FUNCTION_BLOCK FB_ESSMonitoringMCU5001a EXTENDS FB_ESSMonitoringBase
VAR
    //Outputs
    {attribute 'TcLinkTo' := 'TIID^Device 2 (EtherCAT)^KF201 (EK1100)^KF208 (EL2014)^DIG Outputs^Channel 1^Output'}
    bStatusLED AT %Q*: BOOL;
    {attribute 'TcLinkTo' := 'TIID^Device 2 (EtherCAT)^KF201 (EK1100)^KF207 (EL2014)^DIG Outputs^Channel 4^Output'}
    bAcknowledgeLED AT %Q*: BOOL;
    {attribute 'TcLinkTo' := 'TIID^Device 2 (EtherCAT)^KF201 (EK1100)^KF208 (EL2014)^DIG Outputs^Channel 2^Output'}
    bEStopLED AT %Q*: BOOL;
    {attribute 'TcLinkTo' := 'TIID^Device 2 (EtherCAT)^KF201 (EK1100)^KF208 (EL2014)^DIG Outputs^Channel 4^Output'}
    bErrorLED AT %Q*: BOOL;

    //Inputs
    {attribute 'TcLinkTo' := 'TIID^Device 2 (EtherCAT)^KF201 (EK1100)^KF204 (EL1808)^Channel 1^Input'}
    b24VDC1_OK AT %I*: BOOL;
    {attribute 'TcLinkTo' := 'TIID^Device 2 (EtherCAT)^KF201 (EK1100)^KF204 (EL1808)^Channel 2^Input'}
    b24VDC2_OK AT %I*: BOOL;
    {attribute 'TcLinkTo' := 'TIID^Device 2 (EtherCAT)^KF201 (EK1100)^KF204 (EL1808)^Channel 3^Input'}
    b24VDC3_OK AT %I*: BOOL;
    {attribute 'TcLinkTo' := 'TIID^Device 2 (EtherCAT)^KF201 (EK1100)^KF204 (EL1808)^Channel 4^Input'}
    b48VDC1_OK AT %I*: BOOL;
    {attribute 'TcLinkTo' := 'TIID^Device 2 (EtherCAT)^KF201 (EK1100)^KF204 (EL1808)^Channel 5^Input'}
    b48VDC2_OK AT %I*: BOOL;
    {attribute 'TcLinkTo' := 'TIID^Device 2 (EtherCAT)^KF201 (EK1100)^KF204 (EL1808)^Channel 6^Input'}
    b48VDC3_OK AT %I*: BOOL;
    {attribute 'TcLinkTo' := 'TIID^Device 2 (EtherCAT)^KF201 (EK1100)^KF204 (EL1808)^Channel 7^Input'}
    b48VDC4_OK AT %I*: BOOL;
    {attribute 'TcLinkTo' := 'TIID^Device 2 (EtherCAT)^KF201 (EK1100)^KF203 (EL1808)^Channel 1^Input'}
    bFuse1_OK AT %I*: BOOL;
    {attribute 'TcLinkTo' := 'TIID^Device 2 (EtherCAT)^KF201 (EK1100)^KF203 (EL1808)^Channel 2^Input'}
    bFuse2_Error AT %I*: BOOL;
    {attribute 'TcLinkTo' := 'TIID^Device 2 (EtherCAT)^KF201 (EK1100)^KF203 (EL1808)^Channel 3^Input'}
    bFuse3_Error AT %I*: BOOL;
    {attribute 'TcLinkTo' := 'TIID^Device 2 (EtherCAT)^KF201 (EK1100)^KF203 (EL1808)^Channel 4^Input'}
    bFuse4_OK AT %I*: BOOL;
    {attribute 'TcLinkTo' := 'TIID^Device 2 (EtherCAT)^KF201 (EK1100)^KF203 (EL1808)^Channel 5^Input'}
    bFuse5_OK AT %I*: BOOL;
    {attribute 'TcLinkTo' := 'TIID^Device 2 (EtherCAT)^KF201 (EK1100)^KF203 (EL1808)^Channel 6^Input'}
    bFuse6_OK AT %I*: BOOL;
    {attribute 'TcLinkTo' := 'TIID^Device 2 (EtherCAT)^KF201 (EK1100)^KF203 (EL1808)^Channel 7^Input'}
    bFuse7_OK AT %I*: BOOL;
    {attribute 'TcLinkTo' := 'TIID^Device 2 (EtherCAT)^KF201 (EK1100)^KF203 (EL1808)^Channel 8^Input'}
    bFuse8_OK AT %I*: BOOL;
    {attribute 'TcLinkTo' := 'TIID^Device 2 (EtherCAT)^KF201 (EK1100)^KF205 (EL1808)^Channel 1^Input'}
    bEStopReleased AT %I*: BOOL;
    {attribute 'TcLinkTo' := 'TIID^Device 2 (EtherCAT)^KF201 (EK1100)^KF205 (EL1808)^Channel 2^Input'}
    bSTOReleased AT %I*: BOOL;
    {attribute 'TcLinkTo' := 'TIID^Device 2 (EtherCAT)^KF201 (EK1100)^KF206 (EL1808)^Channel 2^Input'}
    bMCBFan_OK AT %I*: BOOL;
    {attribute 'TcLinkTo' := 'TIID^Device 2 (EtherCAT)^KF201 (EK1100)^KF206 (EL1808)^Channel 3^Input'}
    bSPD_OK AT %I*: BOOL;
    {attribute 'TcLinkTo' := 'TIID^Device 2 (EtherCAT)^KF201 (EK1100)^KF206 (EL1808)^Channel 4^Input'}
    bDoorClosed AT %I*: BOOL;
    {attribute 'TcLinkTo' := 'TIID^Device 2 (EtherCAT)^KF201 (EK1100)^KF205 (EL1808)^Channel 8^Input'}
    bAcknowledgeButton AT %I*: BOOL;
    {attribute 'TcLinkTo' := 'TIID^Device 2 (EtherCAT)^KF201 (EK1100)^KF209 (EL3214)^RTD Inputs Channel 1^Value'}
    nTemp1 AT %I*: INT;
    {attribute 'TcLinkTo' := 'TIID^Device 2 (EtherCAT)^KF201 (EK1100)^KF209 (EL3214)^RTD Inputs Channel 2^Value'}
    nTemp2 AT %I*: INT;
    {attribute 'TcLinkTo' := 'TIID^Device 2 (EtherCAT)^KF201 (EK1100)^KF209 (EL3214)^RTD Inputs Channel 3^Value'}
    nTemp3 AT %I*: INT;
    {attribute 'TcLinkTo' := 'TIID^Device 2 (EtherCAT)^KF201 (EK1100)^KF209 (EL3214)^RTD Inputs Channel 4^Value'}
    nTemp4 AT %I*: INT;
    {attribute 'TcLinkTo' := 'TIID^Device 2 (EtherCAT)^Inputs^DevState'}
    nEcMasterDevState AT %I*: UINT;
END_VAR

SUPER^();

METHOD mLink
// Input variables
AcknowledgeButton := bAcknowledgeButton;
EcMasterDevState := nEcMasterDevState;

// Output variables
bAcknowledgeLED := AcknowledgeLED;
bStatusLED := StatusLED;
bEStopLED := EStopLED;
bErrorLED := ErrorLED;

IF iSafetyProvider <> 0 AND_THEN iSafetyProvider.P_ReadFromSafetyController THEN
    _EStopReleased := iSafetyProvider.P_EStopOK;
    _STOReleased := iSafetyProvider.P_STO_OK;
ELSE
    _EStopReleased := bEStopReleased;
    _STOReleased := bSTOReleased;
END_IF;

EStopReleased := _EStopReleased;
END_METHOD

METHOD mSetResetAlarmsLeds
VAR_INST
    index: UINT;
    aDeadBandActive: ARRAY [1..4] OF BOOL;
    nDeadBandTemperature: INT := 3;
    aTemperatureAlarm: ARRAY [1..4] OF BOOL;
END_VAR
mSetReset(stAlarmList := aAlarmList[1], bOk := b24VDC1_OK);
mSetReset(stAlarmList := aAlarmList[2], bOk := b24VDC2_OK);
mSetReset(stAlarmList := aAlarmList[3], bOk := b24VDC3_OK);

mSetReset(stAlarmList := aAlarmList[4], bOk := b48VDC1_OK);
mSetReset(stAlarmList := aAlarmList[5], bOk := b48VDC2_OK);
mSetReset(stAlarmList := aAlarmList[6], bOk := b48VDC3_OK);
mSetReset(stAlarmList := aAlarmList[7], bOk := b48VDC4_OK);

mSetReset(stAlarmList := aAlarmList[8], bOk := bMCBFan_OK);
mSetReset(stAlarmList := aAlarmList[9], bOk := bSPD_OK);
mSetReset(stAlarmList := aAlarmList[10], bOk := bDoorClosed);

mSetReset(stAlarmList := aAlarmList[11], bOk := bFuse1_OK);
mSetReset(stAlarmList := aAlarmList[12], bOk := NOT bFuse2_Error);
mSetReset(stAlarmList := aAlarmList[13], bOk := NOT bFuse3_Error);
mSetReset(stAlarmList := aAlarmList[14], bOk := bFuse4_OK);
mSetReset(stAlarmList := aAlarmList[15], bOk := bFuse5_OK);
mSetReset(stAlarmList := aAlarmList[16], bOk := bFuse6_OK);
mSetReset(stAlarmList := aAlarmList[17], bOk := bFuse7_OK);
mSetReset(stAlarmList := aAlarmList[18], bOk := bFuse8_OK);

mSetReset(stAlarmList := aAlarmList[19], bOk := EStopReleased);

mSetReset(stAlarmList := aAlarmList[24], bOk := NOT bEcMasterError);
mSetReset(stAlarmList := aAlarmList[25], bOk := NOT bSlaveStateNotOP);
mSetReset(stAlarmList := aAlarmList[26], bOk := NOT bSlaveLinkError);
mSetReset(stAlarmList := aAlarmList[27], bOk := NOT bCycleTimeExceeded);
mSetReset(stAlarmList := aAlarmList[28], bOk := NOT bCPUOverloaded);


aTemperatureAlarm[1] :=
    nTemp1 > nMAX_TEMP
    OR (aDeadBandActive[1] AND nTemp1 > (nMAX_TEMP - nDeadBandTemperature));
aDeadBandActive[1] := aTemperatureAlarm[1];
mSetReset(stAlarmList := aAlarmList[20], bOk := NOT aTemperatureAlarm[1]);

aTemperatureAlarm[2] :=
    nTemp2 > nMAX_TEMP
    OR (aDeadBandActive[2] AND nTemp2 > (nMAX_TEMP - nDeadBandTemperature));
aDeadBandActive[2] := aTemperatureAlarm[2];
mSetReset(stAlarmList := aAlarmList[21], bOk := NOT aTemperatureAlarm[2]);

aTemperatureAlarm[3] :=
    nTemp3 > nMAX_TEMP
    OR (aDeadBandActive[3] AND nTemp3 > (nMAX_TEMP - nDeadBandTemperature));
aDeadBandActive[3] := aTemperatureAlarm[3];
mSetReset(stAlarmList := aAlarmList[22], bOk := NOT aTemperatureAlarm[3]);

aTemperatureAlarm[4] :=
    nTemp4 > nMAX_TEMP
    OR (aDeadBandActive[4] AND nTemp4 > (nMAX_TEMP - nDeadBandTemperature));
aDeadBandActive[4] := aTemperatureAlarm[4];
mSetReset(stAlarmList := aAlarmList[23], bOk := NOT aTemperatureAlarm[4]);
END_METHOD

END_FUNCTION_BLOCK

(* stored: Version 1.1.0.1
   POU FB_ESSMonitoringMCU5001a: Id {dc25224c-2805-4e0c-98fe-daa6f852a4e2}, SpecialFunc None
   Method mLink: Id {8f68c928-532a-0184-1c03-483eb2950c4b}
   Method mSetResetAlarmsLeds: Id {1241012c-ae73-450a-94a3-e603ad15f437} *)
